{attribute 'linkalways'} 
{attribute 'no_explicit_call' := 'This FB is a CLASS and must be accessed using methods or properties'}
{attribute 'enable_dynamic_creation'}
FUNCTION_BLOCK Node_F_VN_PutTextExp EXTENDS VisionNode
VAR
    sText : _STRING('');
    ipDestImage : _ITcVnImage;
    nX : _UDINT(1);
    nY : _UDINT(1);
    eFontType : _ETcVnFontType(ETcVnFontType.TCVN_FT_HERSHEY_SIMPLEX);
    fFontScale : _LREAL(1.0);
    aColor : _TcVnVector4_LREAL;
    nThickness : _DINT(1);
    eLineType : _ETcVnLineType(ETcVnLineType.TCVN_LT_4_CONNECTED);
    bBottomLeftOrigin : _BOOL(FALSE);
    hrPrev : _HRESULT(S_OK);
	hresult : _HRESULT(S_OK);
END_VAR

METHOD PUBLIC  Clone : I_Node
VAR
	pNode : POINTER TO Node_F_VN_PutTextExp;
END_VAR
pNode := __NEW(Node_F_VN_PutTextExp);
Clone := pNode^;
END_METHOD

METHOD FB_init : BOOL
VAR_INPUT
	bInitRetains : BOOL; // if TRUE, the retain variables are initialized (warm start / cold start)
	bInCopyCode : BOOL;  // if TRUE, the instance afterwards gets moved into the copy code (online change)
END_VAR
AddParameter('sText', sText);
AddInput('ipDestImage', ipDestImage);
AddParameter('nX', nX);
AddParameter('nY', nY);
AddParameter('eFontType', eFontType);
AddParameter('fFontScale', fFontScale);
AddInput('aColor', aColor);
AddParameter('nThickness', nThickness);
AddParameter('eLineType', eLineType);
AddParameter('bBottomLeftOrigin', bBottomLeftOrigin);
AddInput('hrPrev', hrPrev);
AddOutput('ipDestImage', ipDestImage);
AddOutput('hresult',hresult);
END_METHOD

METHOD PROTECTED OnExecute
hresult.Value := F_VN_PutTextExp(
    sText := sText.Value,
	ipDestImage := ipDestImage.Value,
	nX:= nX.Value,
	nY:= nY.Value,
    eFontType := eFontType.Value,
    fFontScale := fFontScale.Value,
    aColor := aColor.Value,
    nThickness := nThickness.Value,
    eLineType := eLineType.Value,
    bBottomLeftOrigin := bBottomLeftOrigin.Value,
	hrPrev:= hrPrev.Value);
END_METHOD

METHOD PUBLIC PreExecutionCheck
VAR_INPUT
	Check : I_PreExecutionChecks;
END_VAR
Check.IsTrue(ipDestImage.IsValid, 'ipDestImage must contain an image');
Check.IsTrue(nThickness.Value >= 1, 'nThickness must be greater than or equal to 1');
END_METHOD

END_FUNCTION_BLOCK

(* stored: Version 1.1.0.1, ProductVersion 3.1.4024.15
   POU Node_F_VN_PutTextExp: Id {b48937c4-0037-4ecd-9a4b-82b5e011c0db}, SpecialFunc None
   Folder Constructor: Id {7a3cd441-6fd2-47fa-b088-a686e1702798}
   Method Clone: Id {20d9a960-6094-469b-9428-03fd9daeb9ca}
   Method FB_init: Id {122d48a9-f97c-4165-a544-4e92ef93e877}
   Method OnExecute: Id {1f542665-36de-42e3-b31a-28cdbd134b83}
   Method PreExecutionCheck: Id {827e9c01-cb18-48d6-a57e-0f174a28d79e} *)
